(* IEC 61131-3 sources: AXOpen/src/components.mitsubishi.robotics/app/SystemConstants, 2 files *)

(* ---- plc_line_HwIdentifiers.st ---- *)
CONFIGURATION HardwareIDs
    VAR_GLOBAL CONSTANT
        PROFINET_IO_System_HwID : UINT := UINT#256;
        TZ535_PN_HwID : UINT := UINT#260;
        TZ535_PN_In_Out_64_byte_1_In_Out__64_byte_HwID : UINT := UINT#263;
        TZ535_PN_Rack_HwID : UINT := UINT#261;
        TZ535_PN_TZ535_PN_HwID : UINT := UINT#262;
        TZ535_PN_TZ535_PN_2D_TZ535_PNPROFINET_IO_HwID : UINT := UINT#264;
        TZ535_PN_TZ535_PN_profinet_HwID : UINT := UINT#257;
        TZ535_PN_TZ535_PN_profinet_Port_1_HwID : UINT := UINT#258;
        TZ535_PN_TZ535_PN_profinet_Port_2_HwID : UINT := UINT#259;
        plc_line_HwID : UINT := UINT#32;
        plc_line_Rail_0_HwID : UINT := UINT#265;
        plc_line_plc_line_HwID : UINT := UINT#48;
        plc_line_plc_line__plc_line_HwID : UINT := UINT#49;
        plc_line_plc_line_CPU_display_1_HwID : UINT := UINT#54;
        plc_line_plc_line_CPU_exec_unit_1_HwID : UINT := UINT#52;
        plc_line_plc_line_Card_reader_writer_1_HwID : UINT := UINT#51;
        plc_line_plc_line_DP_interface_1_HwID : UINT := UINT#60;
        plc_line_plc_line_LicenseManager_1_HwID : UINT := UINT#42;
        plc_line_plc_line_OPC_UA_1_HwID : UINT := UINT#117;
        plc_line_plc_line_PROFINET_interface_2_HwID : UINT := UINT#72;
        plc_line_plc_line_PROFINET_interface_2_Port_1_HwID : UINT := UINT#73;
        plc_line_plc_line_Virtual_communication_interface_HwID : UINT := UINT#135;
        plc_line_plc_line_plc_line_HwID : UINT := UINT#50;
        plc_line_plc_line_profinet_x1_HwID : UINT := UINT#64;
        plc_line_plc_line_profinet_x1_Port1_HwID : UINT := UINT#65;
        plc_line_plc_line_profinet_x1_Port2_HwID : UINT := UINT#66;

    END_VAR
END_CONFIGURATION

(* ---- plc_line_IoAddresses.st ---- *)
CONFIGURATION IoAddresses
    VAR_GLOBAL
        TZ535_PN_In_Out_64_byte_1_InputAddress_0 AT %IL0: LWORD;
        TZ535_PN_In_Out_64_byte_1_InputAddress_1 AT %IL8: LWORD;
        TZ535_PN_In_Out_64_byte_1_InputAddress_2 AT %IL16: LWORD;
        TZ535_PN_In_Out_64_byte_1_InputAddress_3 AT %IL24: LWORD;
        TZ535_PN_In_Out_64_byte_1_InputAddress_4 AT %IL32: LWORD;
        TZ535_PN_In_Out_64_byte_1_InputAddress_5 AT %IL40: LWORD;
        TZ535_PN_In_Out_64_byte_1_InputAddress_6 AT %IL48: LWORD;
        TZ535_PN_In_Out_64_byte_1_InputAddress_7 AT %IL56: LWORD;
        TZ535_PN_In_Out_64_byte_1_OutputAddress_0 AT %QL0: LWORD;
        TZ535_PN_In_Out_64_byte_1_OutputAddress_1 AT %QL8: LWORD;
        TZ535_PN_In_Out_64_byte_1_OutputAddress_2 AT %QL16: LWORD;
        TZ535_PN_In_Out_64_byte_1_OutputAddress_3 AT %QL24: LWORD;
        TZ535_PN_In_Out_64_byte_1_OutputAddress_4 AT %QL32: LWORD;
        TZ535_PN_In_Out_64_byte_1_OutputAddress_5 AT %QL40: LWORD;
        TZ535_PN_In_Out_64_byte_1_OutputAddress_6 AT %QL48: LWORD;
        TZ535_PN_In_Out_64_byte_1_OutputAddress_7 AT %QL56: LWORD;

    END_VAR
END_CONFIGURATION
